// TwinCAT 3 PLC project CL_ErrorsDatabasePLC
// Title: CL_ErrorsDatabase
// Company: CleanGreens SA
// Author: Martin Coffy and Massimo Lucano
// ProjectVersion: 2.0.4
// Description: class to load error and class messages from SQL database
// ProgramVersion: 3.1.4024.0
// libraries:
//   CL_CleanGreensObjectsLibrary, * (CleanGreens SA)
//   Tc2_Database, * (Beckhoff Automation GmbH)
//   Tc2_DataExchange, * (Beckhoff Automation GmbH)
//   Tc2_Math, * (Beckhoff Automation GmbH)
//   Tc2_Standard, * (Beckhoff Automation GmbH)
//   Tc2_System, * (Beckhoff Automation GmbH)
//   Tc2_Utilities, * (Beckhoff Automation GmbH)
//   Tc3_Database, * (Beckhoff Automation GmbH)
//   Tc3_EventLogger, * (Beckhoff Automation GmbH)
//   Tc3_Module, * (Beckhoff Automation GmbH)
// project tree:
//   DUTs/ Main_STM.TcDUT (not stored), STM_LoadDB.TcDUT, ST_classAndErrorNum.TcDUT, ST_ErrorDBConst.TcDUT (not stored), ST_ParameterValues.TcDUT, ST_SP_ClassReturn.TcDUT, ST_SP_RecordReturn.TcDUT, ST_valToAccess.TcDUT
//   GVLs/ C.TcGVL
//   / PlcTask.TcTTO
//   POUs/Classes_database_connection/ CL_CGSDictionnary.TcPOU, CL_ErrorDB.TcPOU, FB_SP_getClassNameAndIDs.TcPOU, FB_SP_getErrorsMessages.TcPOU

CONFIGURATION CL_ErrorsDatabasePLC
    RESOURCE PLC ON TwinCAT3
        TASK PlcTask(INTERVAL := T#10ms, PRIORITY := 20);
        PROGRAM MAIN WITH PlcTask : MAIN;
    END_RESOURCE
END_CONFIGURATION

// ---- DUTs/STM_LoadDB.TcDUT
{attribute 'qualified_only'}
{attribute 'strict'}
TYPE STM_LoadDB :
(
  
  GetAMSAdress,
	StoreErrorView,
	StoreClassView,
  GenErrorKeys,
	GenClassKeys,
	EndReadingDB
);
END_TYPE

// ---- DUTs/ST_classAndErrorNum.TcDUT
TYPE ST_classAndErrorNum :
	STRUCT
		errorId					: STRING(3);
		classId					: STRING(3);
		telegramSending	: STRING(1);
		hmiErrorShow		: STRING(1);
		instanceNum			: BYTE;
	END_STRUCT
END_TYPE

// ---- DUTs/ST_ParameterValues.TcDUT
TYPE ST_ParameterValues :
STRUCT
	lang: STRING(2);
END_STRUCT
END_TYPE

// ---- DUTs/ST_SP_ClassReturn.TcDUT
TYPE ST_SP_ClassReturn :
STRUCT
	tableId: UDINT;
	classId: STRING(3);
	className: T_MaxString;
	instanceNum: BYTE;
	objDescriptMsg:	T_MaxString;
END_STRUCT
END_TYPE

// ---- DUTs/ST_SP_RecordReturn.TcDUT
TYPE ST_SP_RecordReturn :
STRUCT
	tableId: UDINT;
	//classId: STRING(3);
	errorId: STRING(3);
	severity: BYTE;
	errorMsgShort: T_MaxString;
	errorMsgLong: T_MaxString;
	remediationMsg: T_MaxString;
	telegramSending: STRING(1);
	hmiErrorShow: STRING(1);
END_STRUCT
END_TYPE

// ---- DUTs/ST_valToAccess.TcDUT
TYPE ST_valToAccess :
STRUCT
  	severity: BYTE;
	errorSummary:	T_MaxString;
	errorMessage: T_MaxString;
	remediationMessage: T_MaxString;
	telegramSending: STRING(1);
	hmiErrorShow: STRING(1);
END_STRUCT
END_TYPE

// ---- GVLs/C.TcGVL
// constant to be set in order to describe the greenhouse
// abbreviation GH stands everywhere for Greenhouse
{attribute 'qualified_only'}
VAR_GLOBAL CONSTANT 
  //Errors database constants
  tTimeoutConnectSQLDB_C   : TIME := T#4S;//WAS 15S

  nMaxRecordsDb_C          : UDINT := 1024;
  nMaxUpSize_C             : UDINT := 2048;
  //uiErrorUpSizePowerTwo_C : UDINT := 1024;
  //uiClassUpSizePowerTwo_C : UDINT := 1024;
END_VAR

// ---- POUs/Classes_database_connection/CL_CGSDictionnary.TcPOU
FUNCTION_BLOCK CL_CGSDictionnary
VAR
	bInit	            :	BOOL	:= FALSE;
	
	_usiNbIter_C	    :	USINT;
	_udiSizeKeyArray	:	UDINT;
	
	usiSearchIter     : USINT;
  udiUpId           : UDINT;
  udiDownId         : UDINT;
	
	// Pointer to the keys array to search into
	_udiKeyArray_P	  :	POINTER TO UDINT;	// Access to the keys array with a pointer, limited risks as long as udiUpId and udiDownId are correctly set.
END_VAR

METHOD PUBLIC Init : BOOL
VAR_INPUT
	udiKeyArray_P		  :	POINTER TO UDINT;
	usiNbIter_C			  :	USINT;
	udiSizeKeyArray	  :	UDINT;
END_VAR
VAR
	  udiSizeArCalc   : UDINT;
END_VAR
Init := FALSE;
udiSizeArCalc := LREAL_TO_UDINT(EXPT(2,usiNbIter_C));

IF NOT bInit AND udiKeyArray_P <> 0 AND usiNbIter_C > 0 AND udiSizeArCalc = udiSizeKeyArray THEN
		// Test for the size of the inputs: to check if possible 
		
		// Initialisation of the "constant" values
		_udiKeyArray_P		:= udiKeyArray_P;
		_usiNbIter_C			:= usiNbIter_C;
		_udiSizeKeyArray	:= udiSizeKeyArray;
		
		// Initialisation for the method
		usiSearchIter := usiNbIter_C;
  	udiUpId       := udiSizeKeyArray;
  	udiDownId     := 1;
		bInit := TRUE;
END_IF
END_METHOD

METHOD Search : BOOL
VAR_INPUT
  udiKey_DB	        :	UDINT	:=	0;
END_VAR
VAR_OUTPUT
	udiFoundKeyIndex	:	UDINT;
  bError            : BOOL;
END_VAR
VAR
  udiMidDownId      : UDINT;
  udiMidUpId        : UDINT;
  udiMidUpKey       : UDINT;
  udiMidLowKey      : UDINT;
END_VAR
IF bInit THEN
  Search := FALSE; 
  bError := FALSE;
  udiMidDownId := (udiUpId+udiDownId-1)/2;
  udiMidUpId := udiMidDownId+1;
  udiMidUpKey := _udiKeyArray_P[udiMidUpId-1];	// Correction of index 1, since a pointer to an UINT and not to an array of uint anymore (0-indexing by the TwinCAT syntax, while algorithm meant for an array starting at index 1).
  udiMidLowKey := _udiKeyArray_P[udiMidDownId-1]; // Syntax for pointers of an array: arrayPoint[i] = (arrayPoint + i*size(type))^, with arrayPoint^ the first element of the array
  // Also manage the case when final iter and no case found
  IF udiKey_DB = udiMidLowKey THEN
		udiFoundKeyIndex := udiMidDownId;	// +1 required, since the Pointer index begins at 0, while the corresponding array starts at 1! -- not required anymore!
		usiSearchIter := _usiNbIter_C;
		udiUpId   := _udiSizeKeyArray;
		udiDownId := 1;
    Search := TRUE;
  ELSIF udiMidUpKey = udiKey_DB THEN
		udiFoundKeyIndex := udiMidUpId;	//+1 required, since the Pointer index begins at 0, while the corresponding array starts at 1! -- not required anymore!
		usiSearchIter := _usiNbIter_C;
		udiUpId   := _udiSizeKeyArray;
		udiDownId := 1;
    Search	:= TRUE;
  ELSE 
    IF usiSearchIter > 1 THEN
      IF udiMidLowKey > udiKey_DB THEN
          udiUpId := udiMidDownId;
					usiSearchIter := usiSearchIter-1;
      ELSIF udiMidUpKey < udiKey_DB THEN
          udiDownId := udiMidUpId;
					usiSearchIter := usiSearchIter-1;
      ELSE
				usiSearchIter := _usiNbIter_C;
				udiUpId   := _udiSizeKeyArray;
				udiDownId := 1;
				Search := TRUE;
				bError := TRUE;
      END_IF
    ELSE
			usiSearchIter := _usiNbIter_C;
			udiUpId   := _udiSizeKeyArray;
			udiDownId := 1;
      Search := TRUE;
      bError := TRUE;
    END_IF
  END_IF
END_IF
END_METHOD

END_FUNCTION_BLOCK

// ---- POUs/Classes_database_connection/CL_ErrorDB.TcPOU
{attribute 'enable_dynamic_creation'}
FUNCTION_BLOCK CL_ErrorDB
VAR  
  // Internal variables
  bInit                   :	BOOL	:= FALSE;
  stmMain                 : Main_STM := Main_STM.Init;
	
	// AMS variable
	fbAMSaddrGetter	        :	FB_GetLocalAmsNetId;
  
  // DB related variables
  // langStruct: ST_ParameterValues := (lang := C.sLangErrors);
  dbErrorConnector        : FB_SP_getErrorsMessages;
	dbClassConnector        :	FB_SP_getClassNameAndIDs;
  stmLoadDB               : STM_LoadDB	:= STM_LoadDB.GetAMSAdress;
  udiIndex                : UDINT := 1;
  
  // Size-related variables (previously known)
  _stError_ARP  	        : POINTER TO ARRAY [1..C.nMaxRecordsDb_C] OF ST_SP_RecordReturn;
  _sizeOfstError_AR       : UDINT;
	_stClass_ARP		        : POINTER TO ARRAY [1..C.nMaxRecordsDb_C] OF ST_SP_ClassReturn;
  _sizeOfstClass_AR       : UDINT;
	
  //udiErrorKeys_ARP        : ARRAY[1..C.nMaxUpSize_C] OF UDINT := [C.nMaxUpSize_C(0)];
	//udiClassKeys_ARP		    :	ARRAY[1..C.nMaxUpSize_C] OF UDINT := [C.nMaxUpSize_C(0)];

  udiErrorKeys_ARP        : POINTER TO ARRAY[1..C.nMaxUpSize_C] OF UDINT;
	udiClassKeys_ARP		    :	POINTER TO ARRAY[1..C.nMaxUpSize_C] OF UDINT;
	
	// Dictionnary objects - used to generalised the key search to any type of data structure
	objErrorDict	          :	CL_CGSDictionnary;
	objClassDict	          :	CL_CGSDictionnary;
	
	// Variables containing constants
  _uiClassShiftIndex      : UDINT;
  _uiErrShiftIndex        : UDINT;
  _uiUpSizeErrPowerTwo    : UDINT;
  _uiUpSizeClassPowerTwo  : UDINT;
  _uiErrNumIter           : USINT;
  _uiClassNumIter         : USINT;
	_stConstValues	        :	ST_ErrorDBConst;
	
	// AMS address
	sAMSAdrDbConnect        :	T_AmsNetId;
	stLangMsg               :	ST_ParameterValues	:= (lang := '');	//:= (lang := C.sLangErrors);
END_VAR

METHOD PUBLIC GetClassLongMsg : T_MaxString
VAR_INPUT
	udiIndex	:	UDINT;
END_VAR
if udiIndex > 0 and udiIndex <= _stConstValues.udiClassNumRecord then
  GetClassLongMsg := _stClass_ARP^[udiIndex].objDescriptMsg;
else
  GetClassLongMsg := '';
end_if
END_METHOD

METHOD PUBLIC GetClassShortMsg : T_MaxString
VAR_INPUT
	udiIndex	:	UDINT;
END_VAR
if udiIndex > 0 and udiIndex <= _stConstValues.udiClassNumRecord then
  GetClassShortMsg := _stClass_ARP^[udiIndex].className;
else
  GetClassShortMsg := '';
end_if
END_METHOD

METHOD PUBLIC GetErrorLongMsg : T_MaxString
VAR_INPUT
	udiIndex	:	UDINT;
END_VAR
if udiIndex > 0 and udiIndex <= _stConstValues.udiErrNumRecord then
  GetErrorLongMsg := _stError_ARP^[udiIndex].errorMsgLong;
else
  GetErrorLongMsg := '';
end_if
END_METHOD

METHOD PUBLIC GetErrorRemedMsg : T_MaxString
VAR_INPUT
	udiIndex	:	UDINT;
END_VAR
if udiIndex > 0 and udiIndex <= _stConstValues.udiErrNumRecord then
  GetErrorRemedMsg := _stError_ARP^[udiIndex].remediationMsg;
else
  GetErrorRemedMsg := '';
end_if
END_METHOD

METHOD PUBLIC GetErrorShortMsg : T_MaxString
VAR_INPUT
	udiIndex	:	UDINT;
END_VAR
if udiIndex > 0 and udiIndex <= _stConstValues.udiErrNumRecord then
  GetErrorShortMsg := _stError_ARP^[udiIndex].errorMsgShort;
else
  GetErrorShortMsg := '';
end_if
END_METHOD

METHOD PUBLIC GetNumerics : ST_classAndErrorNum
VAR_INPUT
	udiErrorIndex	:	UDINT;
	udiClassIndex	:	UDINT;
END_VAR
//MPL if the error DB is not loaded or empty or not found, udiClassIndex and/or udiErrorIndex return 0 !!
//MPL write/read to/from the array must be protected against index out of boundaries !!

if udiErrorIndex > 0 and udiErrorIndex <= _stConstValues.udiErrNumRecord then
  GetNumerics.errorId := _stError_ARP^[udiErrorIndex].errorId;
  GetNumerics.hmiErrorShow	:=	_stError_ARP^[udiErrorIndex].hmiErrorShow;
  GetNumerics.telegramSending := _stError_ARP^[udiErrorIndex].telegramSending;
else
  GetNumerics.errorId := '000';
  GetNumerics.hmiErrorShow	:=	'0';
  GetNumerics.telegramSending := '0';  
end_if

if udiClassIndex > 0 and udiClassIndex <= _stConstValues.udiClassNumRecord then
  GetNumerics.classId := _stClass_ARP^[udiClassIndex].classId;
  GetNumerics.instanceNum := _stClass_ARP^[udiClassIndex].instanceNum;
else
  GetNumerics.classId := '000';
  GetNumerics.instanceNum := 0;  
end_if
END_METHOD

METHOD PUBLIC Init : BOOL
VAR_INPUT
  stConstValues   : ST_ErrorDBConst;
END_VAR
VAR
	structSize			: UINT;
	arraySize				: UDINT;
  ind             : UDINT;
END_VAR
_stConstValues := stConstValues;
Init := bInit := FALSE;
IF _stConstValues.udiUsedDB > 0 AND (_stConstValues.udiErrNumRecord > 0) AND (_stConstValues.udiErrNumRecord < C.nMaxRecordsDb_C) AND (_stConstValues.udiClassNumRecord > 0) AND (_stConstValues.udiClassNumRecord < C.nMaxRecordsDb_C) THEN
  _uiUpSizeErrPowerTwo:= nextPower2(_stConstValues.udiErrNumRecord);
  _uiUpSizeClassPowerTwo := nextPower2(_stConstValues.udiClassNumRecord);

  _uiErrShiftIndex := _uiUpSizeErrPowerTwo - _stConstValues.udiErrNumRecord;
  _uiClassShiftIndex := _uiUpSizeClassPowerTwo - _stConstValues.udiClassNumRecord;

  _uiErrNumIter := numIterations(_stConstValues.udiErrNumRecord);
  _uiClassNumIter := numIterations(_stConstValues.udiClassNumRecord);
  
  //Errors DB array allocated in memory from 1..udiErrNumRecord
  structSize := SIZEOF(ST_SP_RecordReturn);
	arraySize := structSize * (_stConstValues.udiErrNumRecord+2);
  _sizeOfstError_AR := structSize * (_stConstValues.udiErrNumRecord+1);
	_stError_ARP := __NEW(BYTE, arraySize);

  //Classes DB array allocated in memory from 1..udiClassNumRecord
  structSize := SIZEOF(ST_SP_ClassReturn);
	arraySize := structSize * (_stConstValues.udiClassNumRecord+2);
  _sizeOfstClass_AR := structSize * (_stConstValues.udiClassNumRecord+1);
	_stClass_ARP := __NEW(BYTE, arraySize);
 
  IF _uiUpSizeErrPowerTwo < C.nMaxUpSize_C AND _uiUpSizeClassPowerTwo < C.nMaxUpSize_C THEN 
    //Errors Keys array allocated in memory from 1.._uiUpSizeErrPowerTwo
    structSize := SIZEOF(UDINT);
    arraySize := structSize * (_uiUpSizeErrPowerTwo+2);
    udiErrorKeys_ARP := __NEW(BYTE, arraySize);
    FOR ind := 1 TO _uiUpSizeErrPowerTwo DO
      udiErrorKeys_ARP^[ind] := 0;
		END_FOR
  
    //Classes Keys array allocated in memory from 1.._uiUpSizeClassPowerTwo
    structSize := SIZEOF(UDINT);
    arraySize := structSize * (_uiUpSizeClassPowerTwo+2);
    udiClassKeys_ARP := __NEW(BYTE, arraySize);
    FOR ind := 1 TO _uiUpSizeClassPowerTwo DO
      udiClassKeys_ARP^[ind] := 0;
		END_FOR
    
    Init := bInit := TRUE;
  END_IF
END_IF
END_METHOD

METHOD PRIVATE nextPower2 : UDINT
VAR_INPUT
  n : UDINT;
END_VAR
VAR
  power : UDINT := 1;
END_VAR
IF (n <= 0) THEN
  nextPower2 := 1;
ELSIF (n AND (n - 1)) = 0 THEN 
  // If n is already a power of 2
  nextPower2 := n;
ELSE

  WHILE (power < n) DO
     //power := SHL(power,1); // Left shift to get the next power of 2}
     power := power * 2;
  END_WHILE
   
  nextPower2 := power;
END_IF
END_METHOD

METHOD PRIVATE numIterations : USINT
VAR_INPUT
  size          : UDINT;
END_VAR
VAR
  log2Size      : LREAL;
  lrNumIter     : LREAL;
  lrNumIterPwr2 : UDINT;
END_VAR
// Calculate the logarithm base 2 of the size
IF size = 1 THEN
	numIterations := 1;	// Explicitly set here, to avoid floating point roundings around 0
ELSIF size > 1 THEN
    log2Size := LN(size) / LN(2.0);
    lrNumIter := LTRUNC(log2Size);
    lrNumIterPwr2 := LREAL_TO_UDINT(EXPT(2,lrNumIter));

    IF size > lrNumIterPwr2 THEN
      numIterations := LREAL_TO_USINT(lrNumIter) + 1;
    ELSE
      numIterations := LREAL_TO_USINT(lrNumIter);
		END_IF
ELSE
    numIterations := 0; // Handle invalid input
END_IF
END_METHOD

METHOD PUBLIC Release : BOOL
VAR_INPUT
END_VAR
bInit := FALSE;
IF _stError_ARP <> 0  THEN 
  __DELETE(_stError_ARP);
END_IF

IF _stClass_ARP <> 0 THEN 
   __DELETE(_stClass_ARP);
END_IF

IF udiErrorKeys_ARP <> 0 THEN 
  __DELETE(udiErrorKeys_ARP);
END_IF

IF udiClassKeys_ARP <> 0 THEN 
  __DELETE(udiClassKeys_ARP);
END_IF
Release := _stError_ARP = 0 AND _stClass_ARP = 0 AND udiErrorKeys_ARP = 0 AND udiClassKeys_ARP = 0;
END_METHOD

METHOD PUBLIC Run : BOOL
VAR_OUTPUT
  bLoadErr:  BOOL;
END_VAR
VAR
  bStillExec: BOOL;
	bAnError: BOOL;
END_VAR
IF NOT bInit THEN
  RETURN;
END_IF
 
Run := FALSE;
bLoadErr := FALSE;

CASE stmLoadDB OF
  STM_LoadDB.GetAMSAdress:	// Useless here, as the previous address was already given
    fbAMSaddrGetter(bExecute := TRUE, tTimeOut := _stConstValues.tAMSTimeout,bBusy => bStillExec, bError => bAnError, AddrString	=> sAMSAdrDbConnect);
      IF NOT bStillExec THEN
        IF bANError THEN
          Run := TRUE;
          bLoadErr := TRUE;
       ELSE
          stLangMsg.lang := _stConstValues.sLanguageForErrors;
          stmLoadDB := STM_LoadDB.StoreErrorView;
        END_IF
      END_IF

  STM_LoadDB.StoreErrorView:
    dbErrorConnector(sAMSNetId := sAMSAdrDbConnect,nDBID := _stConstValues.udiUsedDB, nRecordStartIndex := 0, nLengthRecord := _stConstValues.udiErrNumRecord,tTimeoutIn := _stConstValues.tDBConnectTimeout, sizeRecord := _sizeOfstError_AR, bExecute := TRUE, bBusy => bStillExec, bError => bAnError, stRecord_P := _stError_ARP, stParameterValues := stLangMsg); // tTimeout := T#30S
      IF NOT bStillExec THEN
        IF bANError THEN
          Run := TRUE;
          bLoadErr := TRUE;
        ELSE
          stmLoadDB := STM_LoadDB.StoreClassView;
        END_IF
      END_IF
      
  STM_LoadDB.StoreClassView:
    dbClassConnector(sAMSNetId := sAMSAdrDbConnect, nDBID := _stConstValues.udiUsedDB, nRecordStartIndex := 0, nLengthRecord := _stConstValues.udiClassNumRecord,tTimeoutIn := _stConstValues.tDBConnectTimeout, sizeRecord := _sizeOfstClass_AR, bExecute := TRUE, bBusy => bStillExec, bError => bAnError, stRecord_P := _stClass_ARP);
      IF NOT bStillExec THEN
        IF bANError THEN
          Run := TRUE;
          bLoadErr := TRUE;
        ELSE
          stmLoadDB := STM_LoadDB.GenErrorKeys;
        END_IF
      END_IF
  
  STM_LoadDB.GenErrorKeys:
    udiErrorKeys_ARP^[udiIndex+ _uiErrShiftIndex] := STRING_TO_UDINT(_stError_ARP^[udiIndex].errorId);	// error ID unique for any type of error, no matter the class!
    
    udiIndex := udiIndex + 1;
    IF udiIndex > _stConstValues.udiErrNumRecord THEN
      udiIndex := 1;
      objErrorDict.Init(udiKeyArray_P	:=	udiErrorKeys_ARP,usiNbIter_C := _uiErrNumIter, udiSizeKeyArray := _uiUpSizeErrPowerTwo);
      stmLoadDB := STM_LoadDB.GenClassKeys;
    END_IF
    
STM_LoadDB.GenClassKeys:
    udiClassKeys_ARP^[udiIndex+ _uiClassShiftIndex] := STRING_TO_UDINT(_stClass_ARP^[udiIndex].classId);
    
    udiIndex := udiIndex + 1;
    IF udiIndex > _stConstValues.udiClassNumRecord THEN
      udiIndex := 1;
      objClassDict.Init(udiKeyArray_P	:=	udiClassKeys_ARP,usiNbIter_C := _uiClassNumIter, udiSizeKeyArray := _uiUpSizeClassPowerTwo);
      stmLoadDB := STM_LoadDB.EndReadingDB;  
    END_IF

STM_LoadDB.EndReadingDB:
  Run := TRUE;
  bInit := TRUE;
  bLoadErr := FALSE;
  stmLoadDB := STM_LoadDB.StoreErrorView;
  
END_CASE
END_METHOD

METHOD SearchClassData : BOOL
VAR_INPUT
  classID	:	STRING(3);
END_VAR
VAR_OUTPUT
	udiClassIndex :	UDINT;
  error         : BOOL;
END_VAR
VAR
	bExecEnd      : BOOL;
	foundKey	    :	UDINT;
	uiSafeIter    :	USINT := 0;
END_VAR
REPEAT
	bExecEnd := objClassDict.Search(udiKey_DB := STRING_TO_UDINT(classID),udiFoundKeyIndex => foundKey, bError => error);
	uiSafeIter := uiSafeIter + 1;
	UNTIL (bExecEnd = TRUE) OR (uiSafeIter > _uiClassNumIter)
END_REPEAT

//MPL if the error DB is not loaded or empty or not found, udiClassIndex return 0 !!
// Correction: if an error is found, or that the returned key is zero, then returned class index to zero
IF (error = TRUE) OR (foundKey <= _uiClassShiftIndex) OR (foundKey > _stConstValues.udiClassNumRecord+_uiClassShiftIndex) THEN
	udiClassIndex := 0;
ELSE
	udiClassIndex := foundKey -_uiClassShiftIndex;
END_IF
END_METHOD

METHOD SearchErrorData : BOOL
VAR_INPUT
  errorID	:	STRING(3);
END_VAR
VAR_OUTPUT
	udiErrorIndex	  :	UDINT;
  error           : BOOL;
END_VAR
VAR
	bExecEnd        :	BOOL;
	foundKey	      :	UDINT;
	uiSafeIter      :	USINT := 0;
END_VAR
REPEAT
	bExecEnd := objErrorDict.Search(udiKey_DB := STRING_TO_UDINT(errorID),udiFoundKeyIndex => foundKey, bError => error);
	uiSafeIter := uiSafeIter + 1;
	UNTIL (bExecEnd = TRUE) OR (uiSafeIter > _uiErrNumIter)
END_REPEAT

//MPL if the error DB is not loaded or empty or not found, udiErrorIndex return 0 !!
//Correction: if an error is found, or that the returned key is zero, then returned error index to zero
IF (error = TRUE) OR (foundKey <= _uiErrShiftIndex) OR (foundKey > _stConstValues.udiErrNumRecord+_uiErrShiftIndex) THEN
	udiErrorIndex := 0;
ELSE
	udiErrorIndex := foundKey -_uiErrShiftIndex;
END_IF
END_METHOD

PROPERTY PUBLIC sMsgLang : STRING(2)
GET
sMsgLang := _stConstValues.sLanguageForErrors;
END_GET
END_PROPERTY

METHOD PUBLIC WhichSeverity : BYTE
VAR_INPUT
	udiIndex	: UDINT;
END_VAR
if udiIndex > 0 and udiIndex <= _stConstValues.udiErrNumRecord then
  WhichSeverity := _stError_ARP^[udiIndex].severity;
else
  WhichSeverity := 0;
END_IF
END_METHOD

END_FUNCTION_BLOCK

// ---- POUs/Classes_database_connection/FB_SP_getErrorsMessages.TcPOU
FUNCTION_BLOCK FB_SP_getErrorsMessages
VAR_INPUT
	sAMSNetId	:	T_AmsNetId;
	nDBID	:	UDINT	:= 1;
	nRecordStartIndex: UDINT;
  nLengthRecord:     UDINT;
	tTimeoutIn: TIME;
	bExecute: BOOL;
  stRecord_P: POINTER TO ST_SP_RecordReturn;  // Modified by hand!
  sizeRecord: UDINT;
END_VAR
VAR_OUTPUT
	bBusy: BOOL;
	bError: BOOL;
	ipResult: I_TcMessage;
END_VAR
VAR_IN_OUT
	stParameterValues: ST_ParameterValues;
END_VAR
VAR
	R_TRIG_Execute: R_TRIG;
	nState: INT := 0;
	nErrState: INT;
//	fbSQLDatabase         : FB_SQLDatabaseEvt(sNetID := sAMSNetId, tTimeout := tTimeoutIn);
//	fbSQLStoredProcedure  : FB_SQLStoredProcedureEvt(sNetID := sAMSNetId, tTimeout := tTimeoutIn);
//	fbSQLResult           : FB_SQLResultEvt(sNetID := sAMSNetId, tTimeout := tTimeoutIn);
	fbSQLDatabase         : FB_SQLDatabaseEvt(sNetID := '', tTimeout := C.tTimeoutConnectSQLDB_C);
	fbSQLStoredProcedure  : FB_SQLStoredProcedureEvt(sNetID := '', tTimeout := C.tTimeoutConnectSQLDB_C);
	fbSQLResult           : FB_SQLResultEvt(sNetID := '', tTimeout := C.tTimeoutConnectSQLDB_C);
	arrParaInfo           : ARRAY[0..0] OF ST_SQLSPParameter;
	
END_VAR

CASE nState OF
	0:
		R_TRIG_Execute(CLK:=bExecute);
		IF R_TRIG_Execute.Q THEN
			nState := 1;
			bBusy:=TRUE;
			bError:=FALSE;
			nErrState:=0;
		END_IF
	1:
		IF fbSQLDatabase.Connect(nDBID) THEN
			ipResult:=fbSQLDatabase.ipTcResult;
			IF fbSQLDatabase.bError THEN
				nErrState:=1;
				nState:=255;
			ELSE
				arrParaInfo[0].sParameterName := 'lang';
				arrParaInfo[0].eParameterType := E_SPParameterType.Input;
				arrParaInfo[0].eParameterDataType := E_ColumnType.NChar;
				arrParaInfo[0].nParameterSize := 3;

				nState:= 2;
			END_IF
		END_IF
	2:
		IF fbSQLDatabase.CreateSP('plcGetConfig', ADR(arrParaInfo), SIZEOF(arrParaInfo), ADR(fbSQLStoredProcedure)) THEN
			IF fbSQLDatabase.bError THEN
				nErrState:=2;
				nState:=255;
			ELSE
				nState:=3;
			END_IF
		END_IF
	3:
		IF fbSQLStoredProcedure.ExecuteDataReturn(ADR(stParameterValues), SIZEOF(stParameterValues), ADR(fbSQLResult))THEN
			ipResult:=fbSQLStoredProcedure.ipTcResult;
			IF fbSQLStoredProcedure.bError THEN
				nErrState:=3;
				nState:=255;
			ELSE
				nState:= 4;
			END_IF
		END_IF
	4:
		IF fbSQLResult.Read(nRecordStartIndex, nLengthRecord, stRecord_P, sizeRecord, FALSE, TRUE) THEN
			ipResult:=fbSQLResult.ipTcResult;
			IF fbSQLResult.bError THEN
				nErrState:=4;
				nState:= 255;
			ELSE
				nState:= 5;
			END_IF
		END_IF
	5:
		IF fbSQLStoredProcedure.Release() THEN
			IF fbSQLStoredProcedure.bError THEN
				nErrState:=5;
				nState:=255;
			ELSE
				nState:= 200;
			END_IF
		END_IF
	200:
		IF fbSQLDatabase.Disconnect() THEN
			nState := 0;
			bBusy:= FALSE;
		END_IF
	255:
		bError:= TRUE;
		bBusy:= FALSE;
		IF nErrState > 1 THEN
			nState:=200;
		ELSE
			nState:=0;
		END_IF
END_CASE

END_FUNCTION_BLOCK

// ---- POUs/Classes_database_connection/FB_SP_getClassNameAndIDs.TcPOU
FUNCTION_BLOCK FB_SP_getClassNameAndIDs
VAR_INPUT
	sAMSNetId	:	T_AmsNetId;
	nDBID	:	UDINT	:= 1;
	nRecordStartIndex: UDINT;
	nLengthRecord:	UDINT;
	tTimeoutIn: TIME;
	bExecute: BOOL;
	stRecord_P: POINTER TO ST_SP_ClassReturn;
	sizeRecord: UDINT;
END_VAR
VAR_OUTPUT
	bBusy: BOOL;
	bError: BOOL;
	ipResult: I_TcMessage;
END_VAR
VAR
	R_TRIG_Execute: R_TRIG;
	nState: INT;
	nErrState: INT;
//	fbSQLDatabase: FB_SQLDatabaseEvt(sNetID := sAMSNetId, tTimeout := tTimeoutIn);
//	fbSQLStoredProcedure: FB_SQLStoredProcedureEvt(sNetID := sAMSNetId, tTimeout := tTimeoutIn);
//	fbSQLResult: FB_SQLResultEvt(sNetID := sAMSNetId, tTimeout := tTimeoutIn);
	fbSQLDatabase: FB_SQLDatabaseEvt(sNetID := '', tTimeout := C.tTimeoutConnectSQLDB_C);
	fbSQLStoredProcedure: FB_SQLStoredProcedureEvt(sNetID := '', tTimeout := C.tTimeoutConnectSQLDB_C);
	fbSQLResult: FB_SQLResultEvt(sNetID := '', tTimeout := C.tTimeoutConnectSQLDB_C);
END_VAR

CASE nState OF
	0:
		R_TRIG_Execute(CLK:=bExecute);
		IF R_TRIG_Execute.Q THEN
			nState := 1;
			bBusy:=TRUE;
			bError:=FALSE;
			nErrState:=0;
		END_IF
	1:
		IF fbSQLDatabase.Connect(hDBID := nDBID) THEN
			ipResult:=fbSQLDatabase.ipTcResult;
			IF fbSQLDatabase.bError THEN
				nErrState:=1;
				nState:=255;
			ELSE
				nState:= 2;
			END_IF
		END_IF
	2:
		IF fbSQLDatabase.CreateSP('getClassNameAndIDs', 0, 0, ADR(fbSQLStoredProcedure)) THEN
			IF fbSQLDatabase.bError THEN
				nErrState:=2;
				nState:=255;
			ELSE
				nState:=3;
			END_IF
		END_IF
	3:
		IF fbSQLStoredProcedure.ExecuteDataReturn(0, 0, ADR(fbSQLResult))THEN
			ipResult:=fbSQLStoredProcedure.ipTcResult;
			IF fbSQLStoredProcedure.bError THEN
				nErrState:=3;
				nState:=255;
			ELSE
				nState:= 4;
			END_IF
		END_IF
	4:
		IF fbSQLResult.Read(nRecordStartIndex, nLengthRecord,stRecord_P, sizeRecord, FALSE, TRUE) THEN
			ipResult:=fbSQLResult.ipTcResult;
			IF fbSQLResult.bError THEN
				nErrState:=4;
				nState:= 255;
			ELSE
				nState:= 5;
			END_IF
		END_IF
	5:
		IF fbSQLStoredProcedure.Release() THEN
			IF fbSQLStoredProcedure.bError THEN
				nErrState:=5;
				nState:=255;
			ELSE
				nState:= 200;
			END_IF
		END_IF
	200:
		IF fbSQLDatabase.Disconnect() THEN
			nState := 0;
			bBusy:= FALSE;
		END_IF
	255:
		bError:= TRUE;
		bBusy:= FALSE;
		IF nErrState > 1 THEN
			nState:=200;
		ELSE
			nState:=0;
		END_IF
END_CASE

END_FUNCTION_BLOCK
